// TIA Portal V16 export
// export: Created 2021-08-26T14:43:00.0156319Z, ExportSetting WithDefaults, DisplayName Totally Integrated Automation Portal, DisplayVersion V16, DisplayName TIA Portal Version Control Interface, DisplayVersion V16, DisplayName TIA Portal Openness, DisplayVersion V16, DisplayName STEP 7 Professional, DisplayVersion V16, DisplayName SIMATIC Energy Suite, DisplayVersion V16, DisplayName STEP 7 Safety, DisplayVersion V16, DisplayName WinCC Professional, DisplayVersion V16, DisplayName SIMATIC Visualization Architect, DisplayVersion V16
FUNCTION "MarchaParada" : Void   // FC1, LAD
{ S7_Optimized_Access := 'TRUE' }
VERSION : 0.1
// stored: AutoNumber true, IsIECCheckEnabled false, SetENOAutomatically false, UDAEnableTagReadback false
BEGIN

REGION Network 1
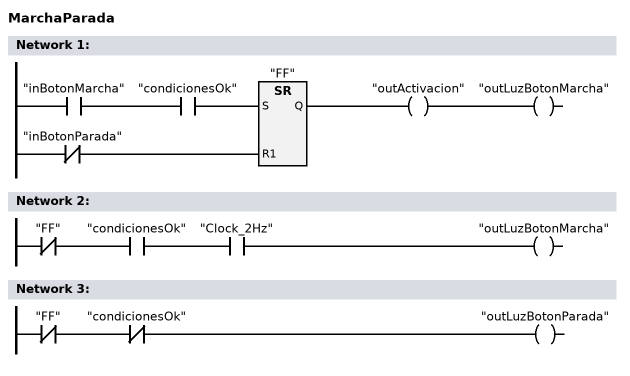
   RUNG wire#powerrail
      Contact( "inBotonMarcha" )
      Contact( "condicionesOk" )
      S_SR(operand := "FF", r1 := wire#w1)
      Coil( "outActivacion" )
      Coil( "outLuzBotonMarcha" )
   END_RUNG
   RUNG wire#powerrail
      I_Contact( "inBotonParada" )
   END_RUNG wire#w1
   // the same network as SCL:
   IF "inBotonMarcha" AND "condicionesOk" THEN
       "FF" := TRUE;   // SR flip-flop
   END_IF;
   IF NOT "inBotonParada" THEN "FF" := FALSE; END_IF;
   "outActivacion" := "FF";
   "outLuzBotonMarcha" := "FF";
END_REGION

REGION Network 2
   RUNG wire#powerrail
      I_Contact( "FF" )
      Contact( "condicionesOk" )
      Contact( "Clock_2Hz" )
      Coil( "outLuzBotonMarcha" )
   END_RUNG
   // the same network as SCL:
   "outLuzBotonMarcha" := NOT "FF" AND "condicionesOk" AND "Clock_2Hz";
END_REGION

REGION Network 3
   RUNG wire#powerrail
      I_Contact( "FF" )
      I_Contact( "condicionesOk" )
      Coil( "outLuzBotonParada" )
   END_RUNG
   // the same network as SCL:
   "outLuzBotonParada" := NOT "FF" AND NOT "condicionesOk";
END_REGION
END_FUNCTION
